ABB RobotStudio station: VoiceCtrlRobot_20221012-214022.rsstn

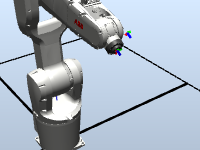
Station VoiceCtrlRobot (saved by RobotStudio 6.8.8307.1040)
Controller VoiceCtrlRobot
  mechanical unit ROB_1: IRB1200_5_90_STD_02, 6 joints, base frame (0, 0, 0) mm
Layout (positions relative to the parent item):
  - IRB1200_5_90_STD_02 [mechanism, from Robots\IRB1200_5_90_STD_02.rslib] at (0, 0, 0) mm; joint values [0, -0.1123, 0.2983, 0, 0.3376, 0] (rad or m)
Targets, tools, work objects and paths stored in the station, written as RAPID:
! task T_ROB1
MODULE Module1
  PERS tooldata toolEquipment:=[TRUE,[[0,0,0],[1,0,0,0]],[1,[0,0,0.001],[1,0,0,0],0,0,0]];
  VAR robtarget homePosition:=[[0,0,0],[1,0,0,0],[0,0,0,0],[9E+09,9E+09,9E+09,9E+09,9E+09,9E+09]];
  VAR speeddata selectedSpeed:=[ 200, 30, 200, 15 ];
  VAR zonedata selectedZone:=[ FALSE, 25, 40, 40, 10, 35, 5 ];
  CONST robtarget Home:=[[521.813982554,0,847.753985316],[0.500000015,0,0.866025395,0],[0,0,0,0],[9E+09,9E+09,9E+09,9E+09,9E+09,9E+09]];
  PROC main()
    MoveJ homePosition,v100,fine,toolEquipment\WObj:=wobj0;
    MoveJ homePosition,v100,fine,toolEquipment\WObj:=wobj0;
    DISTANCE_OP;
    AUTO_OP;
    TOOMATCH_FUNC;
  ENDPROC
  PROC AUTO_OP()
    AUTO_LINEAR_FUNC;
    AUTO_REORIENT_FUNC;
  ENDPROC
  PROC AUTO_LINEAR_FUNC()
    MoveL RelTool(homePosition, disXYZ_m{1},disXYZ_m{2},disXYZ_m{3}, \Rx:= degXYZ_m{1}, \Ry:= degXYZ_m{2}, \Rz:= degXYZ_m{3}),selectedSpeed,selectedZone,toolEquipment\WObj:=wobj0;
  ENDPROC
  PROC AUTO_REORIENT_FUNC()
    MoveL RelTool(homePosition, disXYZ_m{1},disXYZ_m{2},disXYZ_m{3}, \Rx:= degXYZ_m{1}, \Ry:= degXYZ_m{2}, \Rz:= degXYZ_m{3}),selectedSpeed,selectedZone,toolEquipment\WObj:=wobj0;
  ENDPROC
  PROC DISTANCE_OP()
    determined_DISTANCE;
    MoveL RelTool(homePosition,disXYZ_m{1},disXYZ_m{2},disXYZ_m{3} \Rx:= degXYZ_m{1} \Ry:= degXYZ_m{2} \Rz:= degXYZ_m{3} ),v50,fine,toolEquipment\WObj:=wobj0;
    MoveL RelTool(homePosition,disXYZ_m{1},disXYZ_m{2},disXYZ_m{3} \Rx:= degXYZ_m{1} \Ry:= degXYZ_m{2} \Rz:= degXYZ_m{3} ),v50,fine,toolEquipment\WObj:=wobj0;
  ENDPROC
  PROC determined_DISTANCE()
  ENDPROC
  PROC Home_1()
    MoveL Home,v1000,z100,tool0\WObj:=wobj0;
  ENDPROC
  PROC TOOMATCH_FUNC()
  ENDPROC
ENDMODULE

